PROGRAM Qrob_control

VAR_INPUT
	


	torque_set_point AT%Q*:INT;
	torque_enable : BOOL := FALSE;
	enable_torque_out :BOOL;
	torque_decre : REAL :=2;
	
	torque_max_vel : REAL := 200;
	
	actual_torque AT%I*:INT ;
	actual_velocity : REAL;
	done_torqte_lib : BOOL;
	t_aux : INT;
	start_plot : BOOL;
	aux_cu :REAL;
	bthome : BOOL;
	home :	 BOOL;
	reset : bool;
	external : BOOL;
    mover_horario:	BOOL;
	mover_antihorario: BOOL;
	velocidad: REAL := 10 ;
	velocidad_ext: REAL := 100 ;
	set_posicion_mover :INT := 25;
	EnableAxis1 : BOOL := TRUE;
	detener : BOOL;
	mover_abs :BOOL;
	pos_mover_abs :REAL ;
	

	
	
	ajustar_tornillo : BOOL ;
	limite_corriente : REAL := 120;
	torque_relief : BOOL := FALSE;
	tor_on : BOOL;
    tor_val : INT;
		aux_velo : BOOL;
	
END_VAR

VAR
	MC_BufferMode :MC_BufferMode;
	fbPower: MC_Power;
	Axis1Enabled : BOOL;
	actual_position : LREAL;
	//actual_velocity : REAL;
	original_vel :DINT;
	actual_current  :  LREAL;
	position_ok :BOOL;
	
	mov_abs_ok : BOOL;
	max_current : BOOL;
	val_max_current : REAL;
	aux_current : REAL;

	
	MC_Home: MC_HOME;
	MC_ReadActualPosition: MC_ReadActualPosition;
	MC_ReadActualVelocity : MC_ReadActualVelocity;
	MC_ReadParameter_0: MC_ReadParameter;
	MC_MoveVelocity_horario: MC_MoveVelocity;
	MC_MoveVelocity_antiorario: MC_MoveVelocity;
	MC_Stop: MC_Stop;
	MC_Stop2: MC_Stop;
	MC_MoveAbsolute: MC_MoveAbsolute;
    MC_TorqueControl : MC_TorqueControl;
	Ton : TON;
	RS : RS;
	limit_current : limit_current;
	
	
	fuzzy : Subsystem;
	fuzzy_vel : LREAL;
	fuzzy_active : BOOL;
	stop_limit : BOOL;
    MC_ExtSetPointGenEnable : MC_ExtSetPointGenEnable;
	MC_Reset : MC_Reset;
	MC_MoveSuperImposed : MC_MoveSuperImposed;
    FB_CTRL_SETPOINT_GENERATOR : FB_CTRL_SETPOINT_GENERATOR;

	num_ran : LREAL;
	pulse : BOOL:= TRUE;
	PT_b : BOOL;
	DRAND : DRAND;
	pulse1 : pulse_;
	nrand_out : LREAL;
   
	state_move_active : BOOL;	


Max_profile_velocity AT%Q*:UDINT := 314572;
Modes_operation AT%Q*:USINT:= 8;

END_VAR

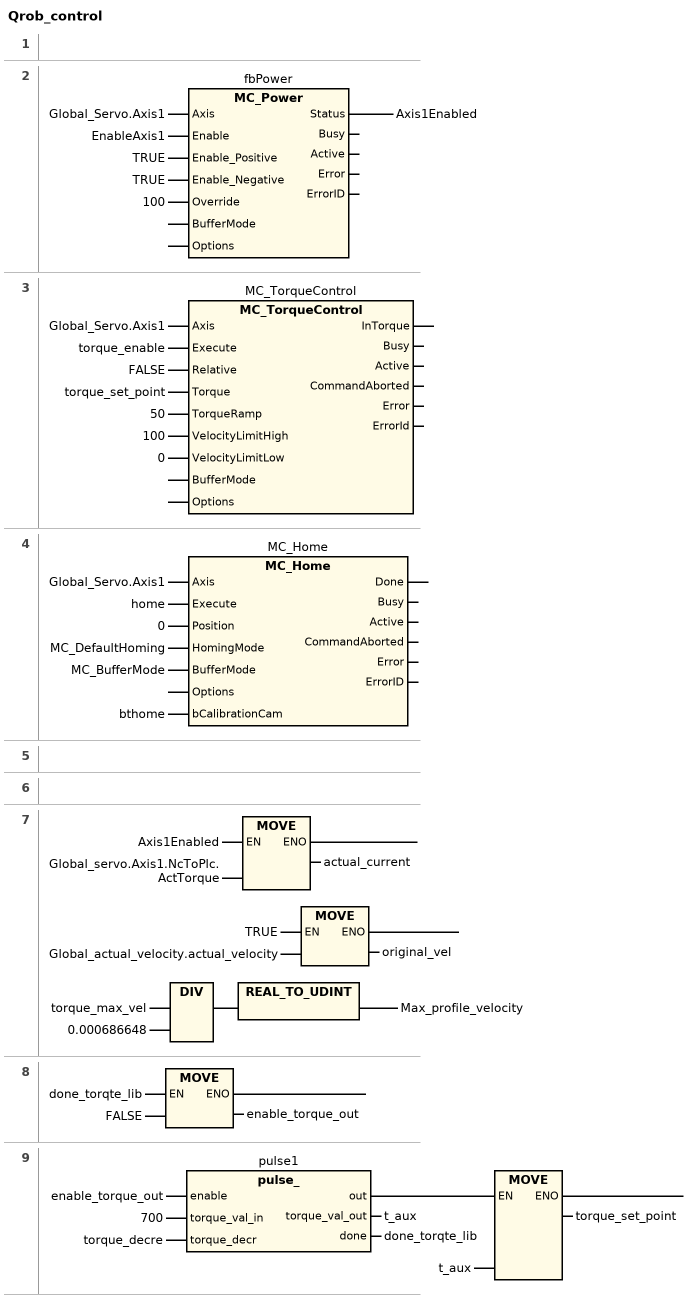
// NETWORK 1

// NETWORK 2
fbPower(
    Axis := Global_Servo.Axis1,
    Enable := EnableAxis1,
    Enable_Positive := TRUE,
    Enable_Negative := TRUE,
    Override := 100); // MC_Power
Axis1Enabled := fbPower.Status;

// NETWORK 3
MC_TorqueControl(
    Axis := Global_Servo.Axis1,
    Execute := torque_enable,
    Relative := FALSE,
    Torque := torque_set_point,
    TorqueRamp := 50,
    VelocityLimitHigh := 100,
    VelocityLimitLow := 0);

// NETWORK 4
MC_Home(
    Axis := Global_Servo.Axis1,
    Execute := home,
    Position := 0,
    HomingMode := MC_DefaultHoming,
    BufferMode := MC_BufferMode,
    bCalibrationCam := bthome);

// NETWORK 5

// NETWORK 6

// NETWORK 7
IF Axis1Enabled THEN actual_current := Global_servo.Axis1.NcToPlc.ActTorque; END_IF
original_vel := Global_actual_velocity.actual_velocity;
Max_profile_velocity := REAL_TO_UDINT(torque_max_vel / 0.000686648);

// NETWORK 8
IF done_torqte_lib THEN enable_torque_out := FALSE; END_IF

// NETWORK 9
pulse1(
    enable := enable_torque_out,
    torque_val_in := 700,
    torque_decr := torque_decre,
    torque_val_out => t_aux,
    done => done_torqte_lib); // pulse_
IF pulse1.out THEN torque_set_point := t_aux; END_IF

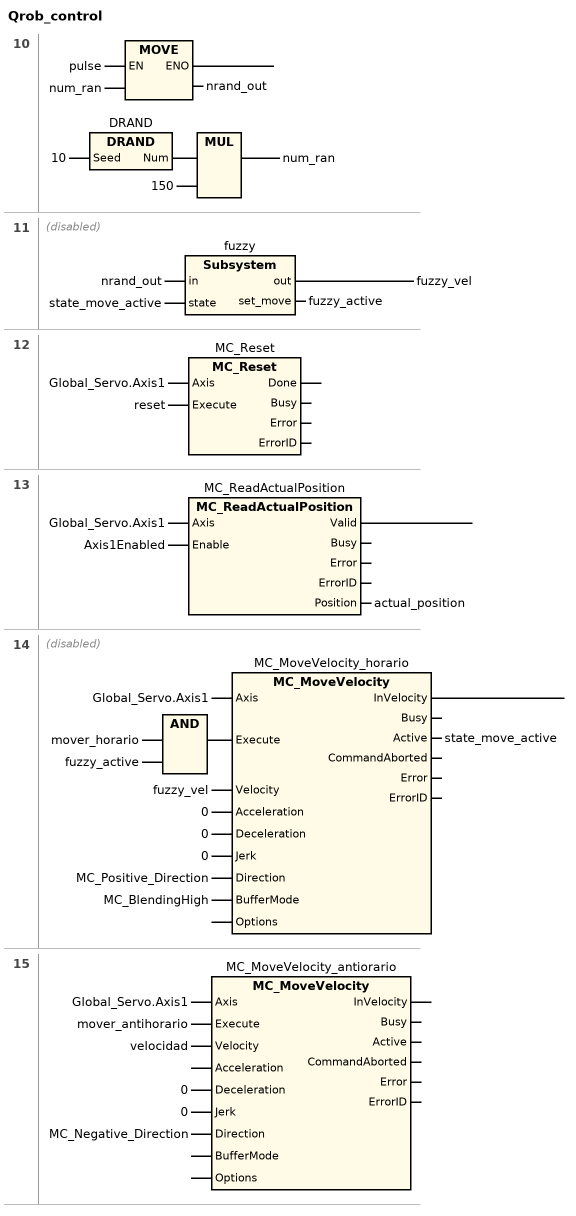
// NETWORK 10
IF pulse THEN nrand_out := num_ran; END_IF
DRAND(Seed := 10);
num_ran := DRAND.Num * 150;

// NETWORK 11 (disabled)
// fuzzy(in := nrand_out, state := state_move_active, set_move => fuzzy_active); // Subsystem
// fuzzy_vel := fuzzy.out;

// NETWORK 12
MC_Reset(Axis := Global_Servo.Axis1, Execute := reset);

// NETWORK 13
MC_ReadActualPosition(Axis := Global_Servo.Axis1, Enable := Axis1Enabled, Position => actual_position);

// NETWORK 14 (disabled)
// MC_MoveVelocity_horario(
//     Axis := Global_Servo.Axis1,
//     Execute := mover_horario AND fuzzy_active,
//     Velocity := fuzzy_vel,
//     Acceleration := 0,
//     Deceleration := 0,
//     Jerk := 0,
//     Direction := MC_Positive_Direction,
//     BufferMode := MC_BlendingHigh,
//     Active => state_move_active); // MC_MoveVelocity

// NETWORK 15
MC_MoveVelocity_antiorario(
    Axis := Global_Servo.Axis1,
    Execute := mover_antihorario,
    Velocity := velocidad,
    Deceleration := 0,
    Jerk := 0,
    Direction := MC_Negative_Direction); // MC_MoveVelocity

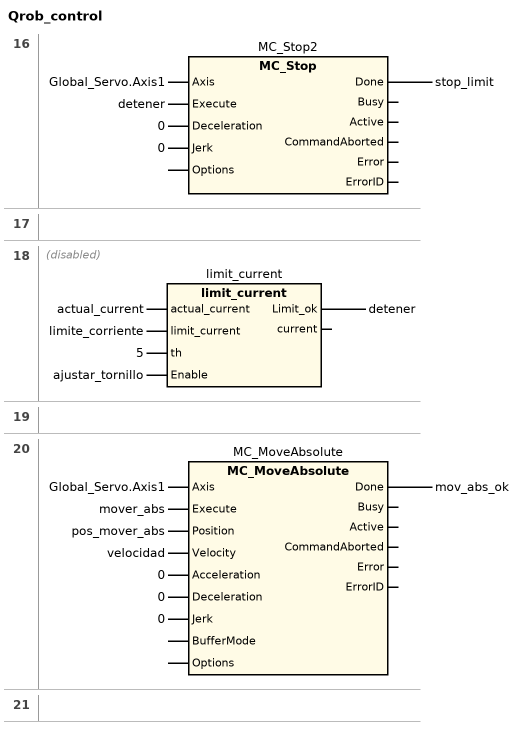
// NETWORK 16
MC_Stop2(Axis := Global_Servo.Axis1, Execute := detener, Deceleration := 0, Jerk := 0); // MC_Stop
stop_limit := MC_Stop2.Done;

// NETWORK 17

// NETWORK 18 (disabled)
// limit_current(
//     actual_current := actual_current,
//     limit_current := limite_corriente,
//     th := 5,
//     Enable := ajustar_tornillo);
// detener := limit_current.Limit_ok;

// NETWORK 19

// NETWORK 20
MC_MoveAbsolute(
    Axis := Global_Servo.Axis1,
    Execute := mover_abs,
    Position := pos_mover_abs,
    Velocity := velocidad,
    Acceleration := 0,
    Deceleration := 0,
    Jerk := 0);
mov_abs_ok := MC_MoveAbsolute.Done;

// NETWORK 21

END_PROGRAM

(* stored: Version 1.1.0.1, ProductVersion 3.1.4024.4
   POU Qrob_control: Id {8c37094b-a5bd-4eb6-9947-3cb2108e38b7}, SpecialFunc None *)
